FUNCTION_BLOCK FB_DMC_MotionControl
VAR_INPUT
	Cmd_Reset			:	BOOL;
	Cmd_Enable			:	BOOL;
	Cmd_MoveAbsolute	:	BOOL;
	Cmd_MoveVelocity	:	BOOL;
	Cmd_MoveRelative	:	BOOL;
	Cmd_JogPositive		:	BOOL;
	Cmd_JogNegative		:	BOOL;
	Cmd_Stop			:	BOOL;
	Cmd_SetPosition		:	BOOL;
	Cfg_Position		:	LREAL;
	Cfg_Velocity		:	LREAL;
	Cfg_Acceleration	:	LREAL;
	Cfg_Deceleration	:	LREAL;
	Cfg_Direction		:	LREAL; //0 = Frw, 1 = Rev, 2 = shortest way
END_VAR
VAR_OUTPUT
END_VAR
VAR
	// Control blocks
	MC_ResetFB 			: Tc3_DriveMotionControl.MC_Reset;
	MC_PowerFB 			: Tc3_DriveMotionControl.MC_Power;
	MC_MoveAbsoluteFB 	: Tc3_DriveMotionControl.MC_MoveAbsolute;
	MC_MoveRelativeFB 	: Tc3_DriveMotionControl.MC_MoveRelative;
	MC_MoveVelocityFB 	: Tc3_DriveMotionControl.MC_MoveVelocity;
	MC_SetPositionFB 	: Tc3_DriveMotionControl.MC_SetPosition;
	MC_HaltFB 			: Tc3_DriveMotionControl.MC_Halt;
	MC_Jog 				: Tc3_DriveMotionControl.MC_Jog;

	// Stepkontrol
	StepControl 		: UINT;
	
	// Enable ONS
	EnableAxisONS		: Tc2_Standard.R_TRIG;
	// Disable ONS
	DisableAxisONS		: Tc2_Standard.R_TRIG;
	
END_VAR
VAR_IN_OUT
	AxisRef		: Tc3_DriveMotionControl.AXIS_REF;
END_VAR

// DMC Simple Motion Control - With standard blocks
// This block is made for inspirational purposes.
// Please make your ovn version that comlies with your / your company´s programming vision
// Version 1.0 - Initial Version
// Version 1.1 - Added MoveRelative & SetPosition
//-----------------------------------------------------------------------------------------

MC_ResetFB(Axis:=AxisRef);// Reset control block
MC_PowerFB(Axis:=AxisRef);// Power/Enable control block
MC_MoveAbsoluteFB(Axis:=AxisRef);// Move To Absolute Position block
MC_MoveVelocityFB(Axis:=AxisRef);// Move Velocity move block
MC_HaltFB(Axis:=AxisRef);// Axis Halt block
MC_Jog(Axis:=AxisRef);// Jog block

EnableAxisONS(CLK:= Cmd_Enable);
DisableAxisONS(CLK:= NOT Cmd_Enable );

// StepControl "case"

CASE Stepcontrol OF

   0: // Holding step
      // Conditions for Reset, Enable, Disable, Start movement, Stop movement, Jog
	  IF Cmd_Reset THEN
		  Cmd_Reset :=0;
		  Stepcontrol :=10;
	  END_IF
	  IF EnableAxisONS.Q THEN
		  Stepcontrol :=20;
	  END_IF
	  IF DisableAxisONS.Q THEN
		  Stepcontrol :=30;
	  END_IF
	  IF Cmd_MoveAbsolute THEN
		  Cmd_MoveAbsolute :=0;
		  Stepcontrol :=40;
	  END_IF
	  IF Cmd_MoveRelative THEN
		  Cmd_MoveRelative :=0;
		  Stepcontrol :=50;
	  END_IF
	  IF Cmd_MoveVelocity THEN
		  Cmd_MoveVelocity :=0;
		  Stepcontrol :=60;
	  END_IF
	  IF Cmd_Stop THEN
		  Cmd_Stop :=0;
		  Stepcontrol :=70;
	  END_IF
	  IF Cmd_JogPositive THEN
		  Stepcontrol :=80;
	  END_IF
	  IF Cmd_JogNegative THEN
		  Stepcontrol :=90;
	  END_IF
 

//---------------------------------RESET---------------------------------
   10: // Reset Axis
       MC_ResetFB.Execute :=TRUE;
       IF MC_ResetFB.Done THEN
          MC_ResetFB.Execute :=FALSE;
          Stepcontrol :=0; // Back to holding step
       END_IF

//---------------------------------POWER---------------------------------
   20: // Enable Axis / Power on Axis
       MC_PowerFB.Enable :=TRUE;
       IF MC_PowerFB.Status THEN
          Stepcontrol :=0; // Back to holding step
       END_IF

   30: // Disable Axis / Removing power from Axis
       MC_PowerFB.Enable :=FALSE;
       IF NOT MC_PowerFB.Status THEN
          Stepcontrol :=0; // Back to holding step
       END_IF

//---------------------------ABSOLUTE MOVEMENT--------------------------------
   40: // Start Absolute Movement
       MC_MoveAbsoluteFB.Execute :=TRUE;
       MC_MoveAbsoluteFB.Velocity := Cfg_Velocity;
       MC_MoveAbsoluteFB.Position := Cfg_Position;
	   MC_MoveAbsoluteFB.Acceleration := Cfg_Acceleration;
	   MC_MoveAbsoluteFB.Deceleration := Cfg_Deceleration;
       IF MC_MoveAbsoluteFB.Active THEN
          MC_MoveAbsoluteFB.Execute :=FALSE;
          Stepcontrol :=45; // Back to holding step
       END_IF

   45:
       IF NOT MC_MoveAbsoluteFB.Done THEN
          Stepcontrol :=0; // Back to holding step
       END_IF
	   
//---------------------------RELATIVE MOVEMENT--------------------------------
   50: // Start Relative Movement
       MC_MoveRelativeFB.Execute :=TRUE;
       MC_MoveRelativeFB.Velocity := Cfg_Velocity;
       MC_MoveRelativeFB.Distance := Cfg_Position;
	   MC_MoveRelativeFB.Acceleration := Cfg_Acceleration;
	   MC_MoveRelativeFB.Deceleration := Cfg_Deceleration;
       IF MC_MoveRelativeFB.Active THEN
          MC_MoveRelativeFB.Execute :=FALSE;
          Stepcontrol :=55; // Back to holding step
       END_IF

   55:
       IF NOT MC_MoveRelativeFB.Done THEN
          Stepcontrol :=0; // Back to holding step
       END_IF

//-----------------------------VELOCITY RUN---------------------------------
   60: // Start Velocity run
       MC_MoveVelocityFB.Execute := TRUE;
       MC_MoveVelocityFB.Velocity := Cfg_Velocity;
	   MC_MoveVelocityFB.Acceleration := Cfg_Acceleration;
	   MC_MoveVelocityFB.Deceleration := Cfg_Deceleration;
	   CASE Cfg_Direction OF
		   0: MC_MoveVelocityFB.Direction := MC_Direction.MC_Positive_Direction;
		   1: MC_MoveVelocityFB.Direction := MC_Direction.MC_Negative_Direction;
		   2: MC_MoveVelocityFB.Direction := MC_Direction.MC_Shortest_Way;
	   END_CASE
       IF MC_MoveVelocityFB.Active THEN
          MC_MoveVelocityFB.Execute := FALSE;
          Stepcontrol :=0; // Back to holding step
       END_IF

   70: // Stop Axis
       MC_HaltFB.Execute :=TRUE;
       IF MC_HaltFB.Done THEN
          MC_HaltFB.Execute :=FALSE;
          Stepcontrol :=0; // Back to holding step
       END_IF

//---------------------------------JOGGING---------------------------------
   80: // Jogging Frw
       MC_Jog.JogForward := TRUE;
       IF MC_Jog.active AND NOT Cmd_JogPositive THEN
          Stepcontrol :=100; // Tilbage til ventestep
       END_IF

   90: // Jogging Rev
       MC_Jog.JogBackwards := TRUE;
       IF MC_Jog.active AND NOT Cmd_JogNegative THEN
          Stepcontrol :=100; // c
       END_IF

   100: // Stop Jog
       MC_Jog.JogForward := FALSE;
       MC_Jog.JogBackwards := FALSE;
       Stepcontrol :=0; // Tilbage til ventestep
	   
//---------------------------SET POSITION--------------------------------
   110: // Set axisposition to xx
       MC_SetPositionFB.Execute :=TRUE;
       MC_SetPositionFB.Position := Cfg_Position;
       IF MC_SetPositionFB.Done THEN 
          MC_SetPositionFB.Execute :=FALSE;
          Stepcontrol :=115; 
       END_IF


END_CASE

END_FUNCTION_BLOCK

(* stored: Version 1.1.0.1, ProductVersion 3.1.4024.14
   POU FB_DMC_MotionControl: Id {3a59ceed-3bdc-4cb1-9fd9-6b66897c30a2}, SpecialFunc None *)
